TYPE ST_InputsPalletMagazine :
STRUCT
	Lift			: ST_LSPM_Inp_LiftSensors;	
	Element 		: ST_LSPM_Inp_Element;	
	CtrlIn			: ST_CtrlInPalletmagazine;
	OpResetSequence	: BOOL;		//Reset sequence operator controled switch/button
END_STRUCT
END_TYPE

(* stored: Version 1.1.0.1, ProductVersion 3.1.4024.4
   DUT ST_InputsPalletMagazine: Id {df0e4b78-350d-4810-8aff-c688a679b5e5} *)
